% RSLogix 500 project 1ST.RSS, saved by version 8.30.00.16 %
PROJECT "UNTITLED"    % processor: Bul.1763 MicroLogix 1100 Series A %

PROGRAM FILES
  LAD 2   6 rungs

DATA FILES
  O0 OUTPUT  4 elements
  I1 INPUT  6 elements
  S2 STATUS  66 elements
  B3 BINARY  1 elements
  T4 TIMER  3 elements
  C5 COUNTER  1 elements
  R6 CONTROL  1 elements
  N7 INTEGER  1 elements
  F8 FLOAT  1 elements

LADDER 2
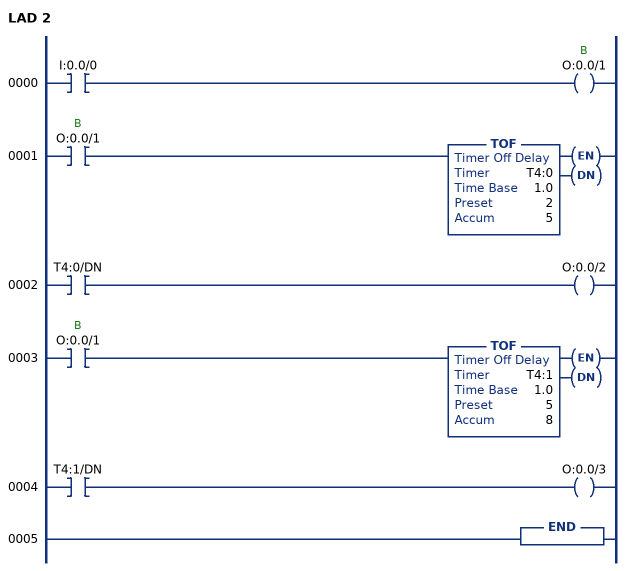
% Rung: 0 %
SOR XIC I:0.0/0 OTE O:0.0/1 EOR
%   O:0.0/1  B %
% Rung: 1 %
SOR XIC O:0.0/1 TOF T4:0 1.0 2 5 EOR
%   O:0.0/1  B %
% Rung: 2 %
SOR XIC T4:0/DN OTE O:0.0/2 EOR
% Rung: 3 %
SOR XIC O:0.0/1 TOF T4:1 1.0 5 8 EOR
%   O:0.0/1  B %
% Rung: 4 %
SOR XIC T4:1/DN OTE O:0.0/3 EOR
% Rung: 5 %
SOR END EOR

DATA TABLE (non-zero values as saved)
DATA T4
% .PRE .ACC %
% T4:0 % 2 5
% T4:1 % 5 8
% T4:2 % 12 12
